FUNCTION TryConvert_REAL_TO_UDINT : BOOL
VAR_INPUT
	in : REAL;
	out : REFERENCE TO UDINT;
END_VAR

IF in > DatatypeLimits.MAX_VALUE_OF_REAL_WHICH_CAN_BE_HELD_IN_A_UDINT THEN
	RETURN;
END_IF

IF in < DatatypeLimits.MIN_VALUE_OF_REAL_WHICH_CAN_BE_HELD_IN_A_UDINT THEN
	RETURN;
END_IF

out := REAL_TO_UDINT(in);
TryConvert_REAL_TO_UDINT := TRUE;

END_FUNCTION

(* stored: Version 1.1.0.1, ProductVersion 3.1.4024.12
   POU TryConvert_REAL_TO_UDINT: Id {c3ab1f1d-9757-4938-9805-4346c85aceef}, SpecialFunc None *)
